FUNCTION_BLOCK Valve (* Composite Function Block Type *)
  (* Standard: 61499-2 *)
  (* Version 0.0, 9/14/2008, Horst Mayer, nxtControl GmbH, template *)
  PACKAGE Main;
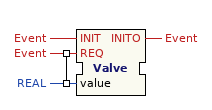
  EVENT_INPUT
    INIT; (* Initialization Request *)
    REQ WITH value; (* Normal Execution Request *)
  END_EVENT
  EVENT_OUTPUT
    INITO; (* Initialization Confirm *)
  END_EVENT
  VAR_INPUT
    value : REAL;
  END_VAR
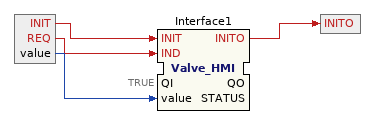
  FBS
    Interface1 : Valve_HMI(QI := TRUE);
  END_FBS
  EVENT_CONNECTIONS
    INIT TO Interface1.INIT;
    REQ TO Interface1.IND;
    Interface1.INITO TO INITO;
  END_CONNECTIONS
  DATA_CONNECTIONS
    value TO Interface1.value;
  END_CONNECTIONS
END_FUNCTION_BLOCK
